(* Schneider Machine Expert - Basic project Lab-06-rodDrive, file version 2.6.0.0 *)
(* ProjectInformations: Name=Lab 6 *)

HARDWARE
  Cpu 0: TM221M16R/G
  EthernetConfiguration: NetworkName=M221, IpAllocationMode=FixedAddress, IpAddress=0.0.0.0, SubnetMask=0.0.0.0
  SerialLineConfiguration: Baud=Baud19200, Parity=ParityEven, DataBits=DataBits8, StopBits=StopBits1, PhysicalMedium=PhysicalMediumRs485, TransmissionMode=TransmissionModeModbusRtu, SlaveId=1, Addressing=SlaveAddressing
  MastTask: UsePeriodScanMode=false, PeriodScan=100
  FastTask: Period=255
  CpuBehavior: StartingMode=StartAsPreviousState, AutoSaveRamOnEeprom=true, WatchdogPeriod=250

SYMBOLS  (address, symbol, comment, settings)
  %M0       STOP
  %I0.0     BTN
  %I0.1     DL
  %Q0.0     RUN

POU Main
  (* SectionNumber=1 *)

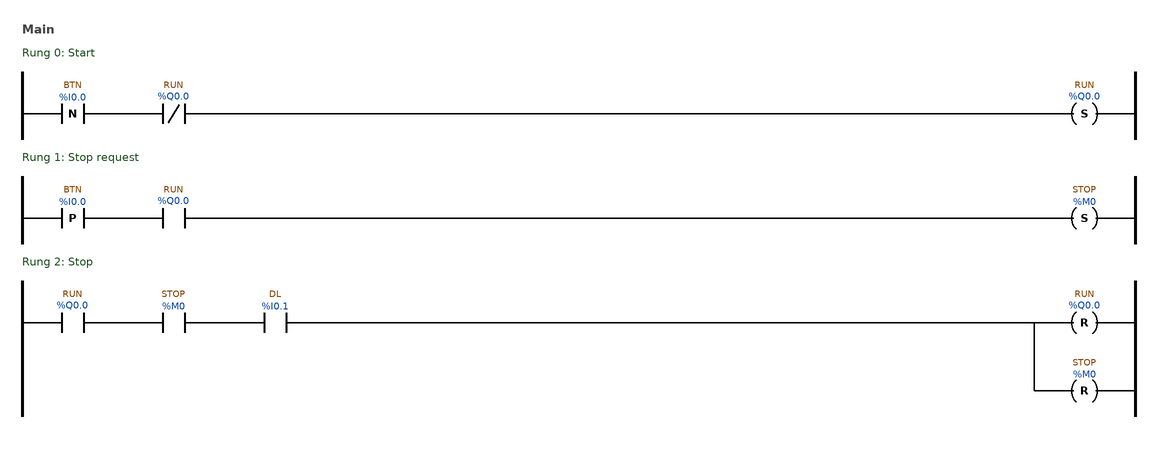

// Rung 0: Start
  LDF %I0.0               (* BTN *)
  ANDN %Q0.0              (* RUN *)
  S %Q0.0                 (* RUN *)
  // as ST:
  //   IF FALLING(BTN) AND NOT RUN THEN RUN := TRUE; END_IF;

// Rung 1: Stop request
  LDR %I0.0               (* BTN *)
  AND %Q0.0               (* RUN *)
  S %M0                   (* STOP *)
  // as ST:
  //   IF RISING(BTN) AND RUN THEN STOP := TRUE; END_IF;

// Rung 2: Stop
  LD %Q0.0                (* RUN *)
  AND %M0                 (* STOP *)
  AND %I0.1               (* DL *)
  R %Q0.0                 (* RUN *)
  R %M0                   (* STOP *)
  // as ST:
  //   _t1 := RUN AND STOP AND DL;
  //   IF _t1 THEN RUN := FALSE; END_IF;
  //   IF _t1 THEN STOP := FALSE; END_IF;
